FUNCTION_BLOCK FB_Valve_4_20A IMPLEMENTS I_Valve
VAR_INPUT
	nOpeningAct AT %I* : REAL;
END_VAR
VAR_OUTPUT
END_VAR
VAR
		//Properties
	bError : BOOL := FALSE;
	fOpeningActual : REAL;
	fOpeningSetpoint : REAL := 0;
	//Raw values
	nOpeningSet AT %Q* : INT;
	//nOpeningAct AT %I* : INT;
END_VAR

PROPERTY Error : BOOL
GET
Error := THIS^.bError;
END_GET
SET
THIS^.bError := Error;
END_SET
END_PROPERTY

PROPERTY OpeningActual : REAL
GET
OpeningActual := THIS^.fOpeningActual;
END_GET
SET
THIS^.fOpeningActual := OpeningActual;
END_SET
END_PROPERTY

PROPERTY OpeningSetpoint : REAL
GET
OpeningSetpoint := THIS^.fOpeningSetpoint;
END_GET
SET
THIS^.fOpeningSetpoint := OpeningSetpoint;
END_SET
END_PROPERTY

METHOD Run
VAR_INPUT
END_VAR
//Read feedback for opening position
fOpeningActual := FC_Current4_20Raw_TO_Percentage(nOpeningAct);

//Write setpoint for opening position
nOpeningSet := FC_Percentage_TO_Current4_20Raw(fOpeningSetpoint);
END_METHOD

END_FUNCTION_BLOCK

(* stored: Version 1.1.0.1, ProductVersion 3.1.4024.3
   POU FB_Valve_4_20A: Id {ce6af1ba-4132-41aa-8a85-00fbaedb61ae}, SpecialFunc None
   Property Error: Id {0bda6983-9627-4240-83f0-dbd93527f96b}
   Get Get: Id {0fe5cdb3-bba7-4923-99c8-d73c1afaa548}
   Set Set: Id {6f61d443-4960-4ded-974a-6d3e5dd78c10}
   Property OpeningActual: Id {fa7c68c9-d6f0-481c-a92e-0d4aeb2e6b8f}
   Get Get: Id {04441374-f5b1-4c60-847c-04925f381feb}
   Set Set: Id {a9331692-55df-472d-ad3d-f775d5027073}
   Property OpeningSetpoint: Id {e361ac6c-ac03-4f95-8661-35094b61ee8e}
   Get Get: Id {ec903a68-f30c-4df2-bb80-8fd8b60c8f22}
   Set Set: Id {405f689d-785a-490e-aed7-1678db059bd7}
   Method Run: Id {fdeed6fd-d672-4a1a-87aa-548838114324} *)
